FUNCTION AnalyzeBatch : ST_ProductStats
VAR_INPUT
	aWeight : ARRAY[1..20] OF REAL;
END_VAR
VAR
	 result : ST_ProductStats;
	 minWeight : REAL;
	 maxWeight : REAL;
END_VAR


FindMinMax(aWeight,  minWeight, maxWeight);

result.averageWeight      := CalculateAverage(aWeight);
result.minWeight     :=   minWeight;
result.maxWeight      :=   maxWeight;
result.defectiveCount  := CountDefects(aWeight);

AnalyzeBatch := result;

END_FUNCTION

(* stored: Version 1.1.0.1, ProductVersion 3.1.4024.16
   POU AnalyzeBatch: Id {5a1dfbf0-8c9c-4042-b221-8f0cce61ceaf}, SpecialFunc None *)
